// TIA Portal project "FactoryIO_Template_S7-1200_V15_V15.1" (V15.1)
// Vorlageprojekt für das Buch mit Zielsystem S7-1200

(* hardware
DEVICE "S7-1200-Station_1"  S7-1200 Station
   slot 0: "Baugruppenträger_0"  Rack  V1.0
   slot 1: "PLC_1"  CPU 1211C DC/DC/DC  6ES7 211-1AE40-0XB0  V4.1
*)

// ===== PLC "PLC_1"  CPU 1211C DC/DC/DC =====

VAR_GLOBAL   // PLC tag table "Standard-Variablentabelle"
   "Tag_1" AT %A0.0 : Bool;
   "Tag_2" AT %E0.0 : Bool;
   "Tag_3" AT %E0.1 : Bool;
END_VAR

VAR_GLOBAL   // PLC tag table "TAG_TABLE_FOR_IO"
   "Start" AT %I0.2 : Bool;   // Start Button
   "Stop" AT %I0.3 : Bool;   // Stop Button
   "Sensor1" AT %I0.4 : Bool;   // For Large box Sensor
   "Sensor2" AT %I0.5 : Bool;   // For small box Sensor
   "Pusher1" AT %Q0.1 : Bool;   // For Large box Pusher
   "Pusher2" AT %Q0.2 : Bool;   // For Large box Pusher
   "Conveyr1" AT %Q0.3 : Bool;
   "Conveyr2" AT %Q0.4 : Bool;
   "Conveyr3" AT %Q0.5 : Bool;
   "Conveyr4" AT %Q0.6 : Bool;
   "Red_Light" AT %Q0.7 : Bool;
   "Green_Light" AT %Q1.0 : Bool;
   "Conveyr5" AT %Q1.1 : Bool;
   "Reset1" AT %I1.0 : Bool;   // Counter Reset for Large Box
   "Reset2" AT %I1.1 : Bool;   // Counter Reset For Small Box
   "Display1" AT %Q1.2 : Bool;
   "Display2" AT %Q1.3 : Bool;
END_VAR

// folder: System blocks/Program resources

DATA_BLOCK "IEC_Timer_0_DB"   // DB1
{ S7_Optimized_Access := 'TRUE' }
AUTHOR : Simatic
FAMILY : IEC
NAME : IEC_TMR
VERSION : 1.0
// stored: InstanceOfName IEC_TIMER
"IEC_TIMER"
BEGIN
END_DATA_BLOCK

DATA_BLOCK "IEC_Timer_0_DB_1"   // DB2
{ S7_Optimized_Access := 'TRUE' }
AUTHOR : Simatic
FAMILY : IEC
NAME : IEC_TMR
VERSION : 1.0
// stored: InstanceOfName IEC_TIMER
"IEC_TIMER"
BEGIN
END_DATA_BLOCK

DATA_BLOCK "IEC_Counter_0_DB_2"   // DB5
{ S7_Optimized_Access := 'TRUE' }
AUTHOR : Simatic
FAMILY : IEC
NAME : CNTR
VERSION : 1.0
// stored: InstanceOfName IEC_COUNTER
"IEC_COUNTER"
BEGIN
END_DATA_BLOCK

DATA_BLOCK "IEC_Counter_0_DB_3"   // DB6
{ S7_Optimized_Access := 'TRUE' }
AUTHOR : Simatic
FAMILY : IEC
NAME : CNTR
VERSION : 1.0
// stored: InstanceOfName IEC_COUNTER
"IEC_COUNTER"
BEGIN
END_DATA_BLOCK

// folder: (top level)

FUNCTION "MHJ-PLC-Lab-Function-S71200" : Void   // FC9000, SCL
{ S7_Optimized_Access := 'TRUE' }
VERSION : 0.1
   VAR_TEMP
      rdTimeReturn : Int;
      outputTime : DTL;
      SyncVal : Byte;
      forVal : Int;
      forVal_2 : Int;
      Value : Byte;
   END_VAR
   VAR CONSTANT
      CompVal : Byte := 16#34;
      Value_01 : Byte := 16#11;
      Value_01_DW : DWord := 16#A165_D992;
      Value_02_DW : DWord := 16#58BE_4401;
   END_VAR
BEGIN

   #Value:=PEEK(area := 16#82,
        dbNumber := 0,
        byteOffset := 511);
   #Value := #Value + 1;

   POKE(area := 16#82,
        dbNumber := 0,
        byteOffset := 511,
        value := #Value);

   POKE(area:=16#81,
        dbNumber:=0,
        byteOffset:=1016,
        value:=#Value_01_DW);
   POKE(area := 16#81,
        dbNumber := 0,
        byteOffset := 1020,
        value := #Value_02_DW);

   POKE(area := 16#81,
        dbNumber := 0,
        byteOffset := 511,
        value := B#16#00);

   FOR #forVal := 0 TO 120 DO
       FOR #forVal_2:=0 TO 10 DO
           #rdTimeReturn:=RD_SYS_T(#outputTime);
           #rdTimeReturn := WR_SYS_T(#outputTime);
           #rdTimeReturn := RD_SYS_T(#outputTime);
           #rdTimeReturn := WR_SYS_T(#outputTime);
       END_FOR;
       #SyncVal:= PEEK(area := 16#81,
                      dbNumber := 0,
                      byteOffset := 511);
       IF #SyncVal = #CompVal THEN
          GOTO M_1;
       END_IF;
   END_FOR;
   RETURN;

   M_1:
   POKE(area := 16#81,
        dbNumber := 0,
        byteOffset := 511,
        value := B#16#0);
END_FUNCTION

ORGANIZATION_BLOCK "Better_Not_To_Modify_This"   // OB1, FBD, ProgramCycle
TITLE = "Main Program Sweep (Cycle)"
{ S7_Optimized_Access := 'TRUE' }
VERSION : 0.1
   VAR_INPUT
      Initial_Call : Bool;   // Initial call of this OB
      Remanence : Bool;   // =True, if remanent data are available
   END_VAR
BEGIN

REGION Network 1: Konnektierungsbaustein für PLC-Lab
   // Im Netzwerk 1 wird der Konnektierungsbaustein für PLC-Lab aufgerufen.
   // Dieser Aufruf darf nicht entfernt werden!
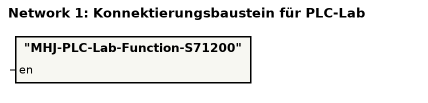
   "MHJ-PLC-Lab-Function-S71200"();
END_REGION

REGION Network 2: Ihr Programm
   // Schreiben Sie ab Netzwerk 2 Ihr Programm
END_REGION
END_ORGANIZATION_BLOCK

ORGANIZATION_BLOCK "Factory_IO_Control_Program"   // OB123, LAD, ProgramCycle
TITLE = "Main Program Sweep (Cycle)"
{ S7_Optimized_Access := 'TRUE' }
VERSION : 0.1
   VAR_INPUT
      Initial_Call : Bool;   // Initial call of this OB
      Remanence : Bool;   // =True, if remanent data are available
   END_VAR
BEGIN

REGION Network 1
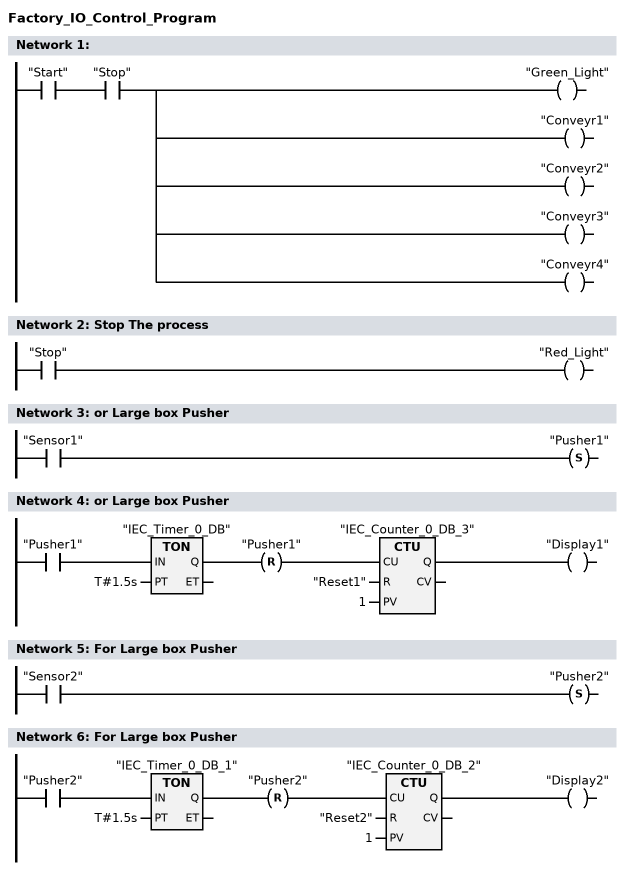
   RUNG wire#powerrail
      Contact( "Start" )
      Contact( "Stop" )
      wire#w1
      Coil( "Green_Light" )
   END_RUNG
   RUNG wire#w1
      Coil( "Conveyr1" )
   END_RUNG
   RUNG wire#w1
      Coil( "Conveyr2" )
   END_RUNG
   RUNG wire#w1
      Coil( "Conveyr3" )
   END_RUNG
   RUNG wire#w1
      Coil( "Conveyr4" )
   END_RUNG
   // the same network as SCL:
   "Green_Light" := "Start" AND "Stop";
   "Conveyr1" := "Green_Light";
   "Conveyr2" := "Green_Light";
   "Conveyr3" := "Green_Light";
   "Conveyr4" := "Green_Light";
END_REGION

REGION Network 2: Stop The process
   RUNG wire#powerrail
      Contact( "Stop" )
      Coil( "Red_Light" )
   END_RUNG
   // the same network as SCL:
   "Red_Light" := "Stop";
END_REGION

REGION Network 3: or Large box Pusher
   RUNG wire#powerrail
      Contact( "Sensor1" )
      S_Coil( "Pusher1" )
   END_RUNG
   // the same network as SCL:
   IF "Sensor1" THEN "Pusher1" := TRUE; END_IF;
END_REGION

REGION Network 4: or Large box Pusher
   "IEC_Timer_0_DB".TON(IN := "Pusher1", PT := T#1.5s);
   IF "IEC_Timer_0_DB".Q THEN "Pusher1" := FALSE; END_IF;
   "IEC_Counter_0_DB_3".CTU(CU := "IEC_Timer_0_DB".Q, R := "Reset1", PV := 1);
   "Display1" := "IEC_Counter_0_DB_3".Q;
END_REGION

REGION Network 5: For Large box Pusher
   RUNG wire#powerrail
      Contact( "Sensor2" )
      S_Coil( "Pusher2" )
   END_RUNG
   // the same network as SCL:
   IF "Sensor2" THEN "Pusher2" := TRUE; END_IF;
END_REGION

REGION Network 6: For Large box Pusher
   "IEC_Timer_0_DB_1".TON(IN := "Pusher2", PT := T#1.5s);
   IF "IEC_Timer_0_DB_1".Q THEN "Pusher2" := FALSE; END_IF;
   "IEC_Counter_0_DB_2".CTU(CU := "IEC_Timer_0_DB_1".Q, R := "Reset2", PV := 1);
   "Display2" := "IEC_Counter_0_DB_2".Q;
END_REGION
END_ORGANIZATION_BLOCK